FUNCTION_BLOCK ABSTRACT FB_Hmi_Component
VAR
	_initialized: BOOL;
END_VAR

PROPERTY PUBLIC ABSTRACT Visibility : BOOL
SET
END_SET
END_PROPERTY

END_FUNCTION_BLOCK

(* stored: Version 1.1.0.1, ProductVersion 3.1.4024.10
   POU FB_Hmi_Component: Id {c3698ac7-38df-4291-b13c-14e193924f32}, SpecialFunc None
   Property Visibility: Id {0496e00a-8a5c-4d8a-aed3-31bf6643fb00}
   Set Set: Id {1bdfbc8a-d582-499a-8c4d-b45e12663124} *)
